FUNCTION_BLOCK SD_Valve
VAR_INPUT
END_VAR
VAR_OUTPUT
    coil : BOOL;
END_VAR
VAR
    _initState : InitState(THIS);
    _autoState : AutoState(THIS);
    _manualState : ManualState(THIS);
    _state : I_SD_ValveState := _initState;
    _stateName : STRING;
END_VAR

_state.RUN();
_stateName := _state.StateName;

METHOD CloseValve : BOOL
CloseValve := _state.Close();
END_METHOD

METHOD GoToAutoState
_state := _autoState;
END_METHOD

METHOD GoToInitState
_state := _initState;
END_METHOD

METHOD GoToManualState
_state := _ManualState;
END_METHOD

METHOD OpenValve : BOOL
OpenValve := _state.Open();
END_METHOD

END_FUNCTION_BLOCK

(* stored: Version 1.1.0.1, ProductVersion 3.1.4024.12
   POU SD_Valve: Id {dfbd4953-2f88-4651-8be7-80f3e286c22c}, SpecialFunc None
   Method CloseValve: Id {67c8e181-db4b-47ab-8f6b-24c02f0f7752}
   Method GoToAutoState: Id {4c78cffb-48b2-4393-b27f-ae1f82ca44ec}
   Method GoToInitState: Id {b94662f6-2200-4c1c-8721-06c0c6ad3338}
   Method GoToManualState: Id {9bcfc7b2-1821-4886-925e-46c8f81bc609}
   Method OpenValve: Id {4120ee58-4a97-48d2-8314-ffb140277f52} *)
